{attribute 'pack_mode' := '1'}
TYPE ST_OdriveSetInputVel :
STRUCT
    rInputVel : REAL;
    rInputTorqueFF : REAL;
END_STRUCT
END_TYPE

(* stored: Version 1.1.0.1
   DUT ST_OdriveSetInputVel: Id {719cd2a6-659d-4733-be04-861dd71e2ba8} *)
